FUNCTION_BLOCK PID
VAR_INPUT
END_VAR
VAR_OUTPUT
END_VAR
VAR
	FB_CTRL_PID: FB_CTRL_PID;
	stCTRL_PID_PARAMS: ST_CTRL_PID_PARAMS;
	Init : BOOL:=TRUE;
	fManSyncValue : LREAL;
	fOut : LREAL;
END_VAR


IF Init THEN
	stCTRL_PID_PARAMS.tCtrlCycleTime 	:= T#10MS;
	stCTRL_PID_PARAMS.tTaskCycleTime 	:= T#10MS;
	stCTRL_PID_PARAMS.fKp				:= 15.0;
	stCTRL_PID_PARAMS.tTn				:= T#20S;
	stCTRL_PID_PARAMS.tTv				:= T#0S;
	stCTRL_PID_PARAMS.tTd				:= T#0S;
	stCTRL_PID_PARAMS.fOutMaxLimit		:= 1000;
	stCTRL_PID_PARAMS.fOutMinLimit		:= -1000;
	
	Init := FALSE;
END_IF

FB_CTRL_PID(
	fSetpointValue:= INT_TO_LREAL(SetPoint), 
	fActualValue:= INT_TO_LREAL(LevelMeter), 
	fManSyncValue:= fManSyncValue, 
	bSync:= FALSE, 
	eMode:= eCTRL_MODE_ACTIVE, 
	bHold:= FALSE, 
	fOut=> fOut, 
	bARWactive=> , 
	eState=> , 
	eErrorId=> , 
	bError=> , 
	stParams:= stCTRL_PID_PARAMS);
	
IF fOut >= 0 THEN
	FillValve := LREAL_TO_INT(fOut);
	DischargeValve := 0;
ELSE
	FillValve := 0;
	DischargeValve := ABS(LREAL_TO_INT(fOut));
END_IF

END_FUNCTION_BLOCK

(* stored: Version 1.1.0.1, ProductVersion 3.1.4024.6
   POU PID: Id {6cbe4950-e171-4e3b-a7a3-1d36991c23a2}, SpecialFunc None *)
